FUNCTION_BLOCK NonlinearController
VAR_INPUT
	robotPose				: RobotPoseSimple;		// Actual robot pose [x, y, theta] in global frame
	robotPoseRef			: RobotPoseSimple;		// Reference robot pose [x, y, theta] in global frame
	robotVelocitiesRef		: RobotPoseSimple;		// Reference robot velocites [vX, vY, omega] in global frame
	vRef					: LREAL;				// Reference linear velocity along path
	enable					: BOOL;
END_VAR

VAR_OUTPUT
	vX						: LREAL;				// Output reference x-velocity in global frame for low-level controller
	vY						: LREAL;				// Output reference y-velocity in global frame for low-level controller
	omega					: LREAL;				// Output refernce angular velocity for low-level controller
	reachedReference		: BOOL;
END_VAR

VAR
	k1, k2, k3				: LREAL;				// Control parameters
	xE, yE, thetaE			: LREAL;				// Robot pose error
	u1, u2					: LREAL;				// Control variables
	xRef, yRef, thetaRef	: LREAL;				// 
	omegaRef				: LREAL;				//
	xAct, yAct, thetaAct	: LREAL;	
	vTransMax				: LREAL := 0.93;
	vRotMax					: LREAL := 1.57;
	positionTolerance		: LREAL := 0.002;
	orientationTolerance	: LREAL := 0.01;
	vRef					: LREAL;				// Reference linear velocity along path
END_VAR

// Reset effective control varibales
vX := 0;
vY := 0;
omega := 0;

k1 := 10;
k3 := 1;

IF enable THEN
	xRef := robotPoseRef.x / 1000;
	yRef := robotPoseRef.y / 1000;
	thetaRef := robotPoseRef.theta;
	omegaRef := robotVelocitiesRef.theta;
	xAct := robotPose.x / 1000;
	yAct := robotPose.y / 1000;
	thetaAct := robotPose.theta;
	
	vRef := SQRT(EXPT(xRef, 2) + EXPT(yRef, 2));

	// Suggested value for k2
	k2 := 2 * ABS(vRef) * SQRT(k3);
	
	// Control errors in mobile reference frame
	xE := COS(thetaAct) * (xRef - xAct) + SIN(thetaAct) * (yRef - yAct);
	yE := -SIN(thetaAct) * (xRef - xAct) + COS(thetaAct) * (yRef - yAct);
	thetaE := -(thetaRef - thetaAct);
	
	// Control law
	u2 := -k2 * thetaE + k3 * vRef * yE * SI(thetaE);
	u1 := vRef * (COS(thetaE) - 1) + yE * (omegaRef + u2) + k1 * xE;
	
	// Write effective control variables
	vX := (u1 + vRef) * COS(thetaAct);
	vY := (u1 + vRef) * SIN(thetaAct);
	omega := u2 + omegaRef;
	
	// Limit effective control variables
	IF (vX > vTransMax) THEN
		vX := vTransMax;
	ELSIF (vX < - vTransMax) THEN
		vX := - vTransMax;
	END_IF
	
	IF (vY > vTransMax) THEN
		vY := vTransMax;
	ELSIF (vY < - vTransMax) THEN
		vY := - vTransMax;
	END_IF
	
	IF (omega > vRotMax) THEN
		omega := vRotMax;
	ELSIF (omega < - vRotMax) THEN
		omega := - vRotMax;
	END_IF
	
	reachedReference := (SQRT(EXPT(xE, 2) + EXPT(yE, 2)) < positionTolerance) AND (ABS(thetaE) < orientationTolerance);
	
	// Scale back to mm / s
	vX := vX * 1000;
	vY := vY * 1000;
END_IF

METHOD reset : BOOL
VAR_INPUT
END_VAR
reachedReference := FALSE;
END_METHOD

END_FUNCTION_BLOCK

(* stored: Version 1.1.0.1, ProductVersion 3.1.4024.11
   POU NonlinearController: Id {5ff6b0a7-4be6-429b-a60b-d6bad624dc52}, SpecialFunc None
   Method reset: Id {857ea841-3f2b-49f1-aa5c-fcb1987df13c} *)
